// TIA Portal project "Toggle Butonu Kullanımı Konvenyör Bandını Hızının Ayarlaması" (V15.1)

(* hardware
DEVICE "PC-System_1"  SIMATIC PC station
   slot 0: "SIMATIC PC station"  Rail  SIMATIC PC-Station  V1.0
      slot 125: "Stationmanager"  Station_Manager  V6.0.4
   slot 1: "HMI_RT_1"  WinCC RT Advanced  6AV2 104-0xxxx-xxxx  15.1.0.0
      slot 33792: "Host interface"  Host interface
   slot 2: "IE general_1"  IE General  IE_CP  V8.2.0
DEVICE "S7-1200 station_1"  S7-1200 Station
   slot 0: "Rack_0"  S7-1200 Rack  Rack  V1.0
   slot 1: "PLC_1"  CPU 1212C DC/DC/DC  6ES7 212-1AE40-0XB0  V4.2
*)

// ===== PLC "PLC_1"  CPU 1212C DC/DC/DC =====

VAR_GLOBAL   // PLC tag table "Default tag table"
   "stop" AT %M5.0 : Bool;
   "start" AT %M5.1 : Bool;
   "sistem_devrede" AT %M5.2 : Bool;
   "konvenyor_calıs" AT %M5.3 : Bool;
   "hızlandır_butonu" AT %M5.4 : Bool;
   "yavaslandir_butonu" AT %M5.5 : Bool;
   "anlık_hız" AT %QW30 : Int;
   "poz_ken" AT %M10.3 : Bool;
   "neg_ken" AT %M10.4 : Bool;
   "uyari_lambasi" AT %Q0.0 : Bool;
END_VAR

VAR_GLOBAL   // PLC tag table "hmi_tags"
   "HMI_toggle" AT %M5.7 : Bool;
END_VAR

ORGANIZATION_BLOCK "Main"   // OB1, LAD, ProgramCycle
TITLE = "Main Program Sweep (Cycle)"
{ S7_Optimized_Access := 'TRUE' }
VERSION : 0.1
   VAR_INPUT
      Initial_Call : Bool;   // Initial call of this OB
      Remanence : Bool;   // =True, if remanent data are available
   END_VAR
   VAR_TEMP   // added for the SCL form of the ladder/FBD networks
      _w1 : Bool;
   END_VAR
BEGIN

REGION Network 1: HMI START
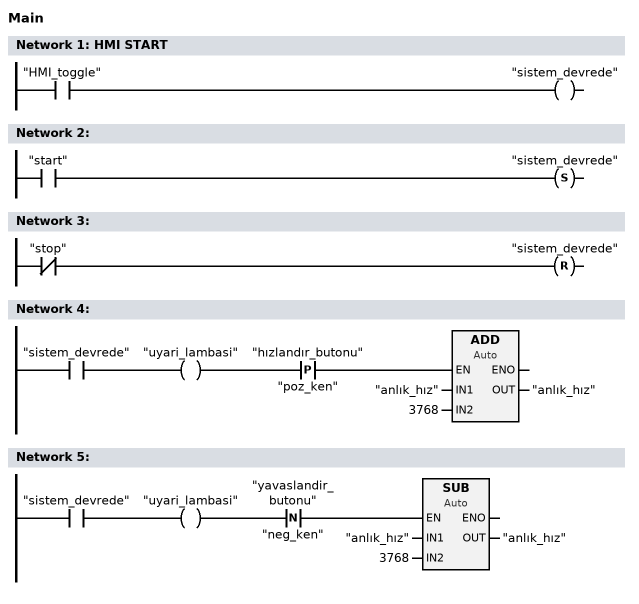
   RUNG wire#powerrail
      Contact( "HMI_toggle" )
      Coil( "sistem_devrede" )
   END_RUNG
   // the same network as SCL:
   "sistem_devrede" := "HMI_toggle";
END_REGION

REGION Network 2
   RUNG wire#powerrail
      Contact( "start" )
      S_Coil( "sistem_devrede" )
   END_RUNG
   // the same network as SCL:
   IF "start" THEN "sistem_devrede" := TRUE; END_IF;
END_REGION

REGION Network 3
   RUNG wire#powerrail
      I_Contact( "stop" )
      R_Coil( "sistem_devrede" )
   END_RUNG
   // the same network as SCL:
   IF NOT "stop" THEN "sistem_devrede" := FALSE; END_IF;
END_REGION

REGION Network 4
   RUNG wire#powerrail
      Contact( "sistem_devrede" )
      Coil( "uyari_lambasi" )
      P_Contact(operand := "hızlandır_butonu", bit := "poz_ken")
      Add(in1 := "anlık_hız", in2 := 3768, out => "anlık_hız")
   END_RUNG
   // the same network as SCL:
   "uyari_lambasi" := "sistem_devrede";
   #_w1 := "sistem_devrede" AND "hızlandır_butonu" AND NOT "poz_ken";   // rising edge of "hızlandır_butonu"
   "poz_ken" := "hızlandır_butonu";
   IF #_w1 THEN "anlık_hız" := "anlık_hız" + 3768; END_IF;
END_REGION

REGION Network 5
   RUNG wire#powerrail
      Contact( "sistem_devrede" )
      Coil( "uyari_lambasi" )
      N_Contact(operand := "yavaslandir_butonu", bit := "neg_ken")
      Sub(in1 := "anlık_hız", in2 := 3768, out => "anlık_hız")
   END_RUNG
   // the same network as SCL:
   "uyari_lambasi" := "sistem_devrede";
   #_w1 := "sistem_devrede" AND NOT "yavaslandir_butonu" AND "neg_ken";   // falling edge of "yavaslandir_butonu"
   "neg_ken" := "yavaslandir_butonu";
   IF #_w1 THEN "anlık_hız" := "anlık_hız" - 3768; END_IF;
END_REGION
END_ORGANIZATION_BLOCK

(* ===== HMI "HMI_RT_1" =====
system functions are stored by id; their names below are inferred from use
connection "HMI_Connection_1": ETHERNET, S7_1200_OMS

HMI tags "Default tag table"
   "HMI_toggle" : Bool = PLC HMI_toggle AT %M5.7, 100 ms
   "HMI_start" : Bool = PLC start AT %M5.1, 100 ms
   "HMI_stop" : Bool = PLC stop AT %M5.0, 100 ms
   "HMI_azalt" : Bool = PLC yavaslandir_butonu AT %M5.5, 1 s
   "HMI_arttir" : Bool = PLC hızlandır_butonu AT %M5.4, 1 s

screen "Screen_1" 1024x768
   Button "Button_1" at 88,125 size 142x153; TextOff 'TOGGLE BUTONU'
      on Press: InvertBit("HMI_toggle")
   Button "Button_2" at 282,70 size 106x120; TextOff 'Text'; PictureOff "Up_Arrow"
      on Press: SetBit("HMI_arttir")
      on Release: ResetBit("HMI_azalt")
      ObjectEnable <- "HMI_arttir"
   Button "Button_3" at 285,244 size 106x120; TextOff 'Text'; PictureOff "Down_Arrow"
      on Release: ResetBit("HMI_azalt")
      on Press: SetBit("HMI_azalt")
      Appearance <- "HMI_azalt"
   TextField "Text field_1" at 273,26 size 506x43; Text 'KONVENYOR BANDI HIZLANDIRMA'
   Button "Button_4" at 482,280 size 96x32; TextOff 'START'
      on Press: SetBit("HMI_start")
   Button "Button_5" at 602,280 size 96x32; TextOff 'STOP'
      on Press: ResetBit("HMI_stop")
      on Release: SetBit("HMI_stop")
*)